// TIA Portal V17 export
// export: Created 2026-04-13T11:12:41.7444866Z, ExportSetting WithDefaults, DisplayName Totally Integrated Automation Portal, DisplayVersion V17 Update 4, DisplayName TIA Portal Openness, DisplayVersion V17 Update 4, DisplayName TIA Portal Version Control Interface, DisplayVersion V17, DisplayName SINAMICS Startdrive Advanced, DisplayVersion V17, DisplayName SINAMICS Startdrive G130, G150, S120, S150, SINAMICS MV, S210, DisplayVersion V17, DisplayName SINAMICS Startdrive G110M, G120, G120C, G120D, G120P, G115D, DisplayVersion V17, DisplayName STEP 7 Professional, DisplayVersion V17 Update 4, DisplayName STEP 7 Safety, DisplayVersion V17, DisplayName WinCC Professional, DisplayVersion V17 Update 4
FUNCTION_BLOCK "A9-循环下料控制"   // FB15, SCL
{ S7_Optimized_Access := 'TRUE' }
VERSION : 0.1
// stored: AutoNumber true, IsIECCheckEnabled false, IsRetainMemResEnabled false, MemoryReserve 100, SetENOAutomatically false, UDAEnableTagReadback false
   VAR_INPUT
      下料启动开关 : Bool;
      上卸料阀工作时间 : Real;
      上卸料阀关闭时间 : Real;
      下卸料阀工作时间 : Real;
      下卸料阀关闭时间 : Real;
   END_VAR
   VAR_OUTPUT
      上阀实际工作时间 : Real;
      上阀实际停止时间 : Real;
      下阀实际工作时间 : Real;
      下阀实际停止时间 : Real;
   END_VAR
   VAR_IN_OUT
      上下料阀 : Bool;
      下下料阀 : Bool;
      振动筛 : Bool;
   END_VAR
   VAR
      上下料阀实际工作时间 : Time;
      上下料阀实际停止时间 : Time;
      下下料阀实际工作时间 : Time;
      下下料阀实际停止时间 : Time;
      循环间隔实际时间 : Time;
      上阀打开辅助 : Bool;
      上阀关闭辅助 : Bool;
      下阀打开辅助 : Bool;
      下阀关闭辅助 : Bool;
      循环工作时间延时 { S7_SetPoint := 'True'} : TON_TIME;
      上阀打开检测1 { S7_SetPoint := 'True'} : R_TRIG;
      上阀打开检测2 { S7_SetPoint := 'True'} : R_TRIG;
      上阀工作时间延时 { S7_SetPoint := 'True'} : TON_TIME;
      上阀停止时间延时 { S7_SetPoint := 'True'} : TON_TIME;
      下阀工作时间延时 { S7_SetPoint := 'True'} : TON_TIME;
      下阀停止时间延时 { S7_SetPoint := 'True'} : TON_TIME;
      下阀打开检测 { S7_SetPoint := 'True'} : R_TRIG;
   END_VAR
BEGIN

   #上下料阀实际工作时间 := DINT_TO_TIME(REAL_TO_DINT(#上卸料阀工作时间*1000.0));
   #上下料阀实际停止时间 := DINT_TO_TIME(REAL_TO_DINT(#上卸料阀关闭时间 * 1000.0));
   #下下料阀实际工作时间 := DINT_TO_TIME(REAL_TO_DINT(#下卸料阀工作时间 * 1000.0));
   #下下料阀实际停止时间 := DINT_TO_TIME(REAL_TO_DINT(#下卸料阀关闭时间 * 1000.0));

   #上阀打开检测1(CLK:=#下料启动开关);


   IF #上阀打开检测1.Q THEN
       #上阀打开辅助 := TRUE;
   END_IF;


   #上阀工作时间延时.TON(IN:=#上阀打开辅助 AND #下料启动开关 AND NOT #下阀停止时间延时.Q,PT:=#上下料阀实际工作时间);

   #上阀停止时间延时.TON(IN:=#上阀工作时间延时.Q,PT:=#上下料阀实际停止时间);

   #下阀工作时间延时(IN:=#上阀工作时间延时.Q AND #上阀停止时间延时.Q,PT:=#下下料阀实际工作时间);

   #下阀停止时间延时(IN :=#上阀工作时间延时.Q AND #上阀停止时间延时.Q AND  #下阀工作时间延时.Q,PT := #下下料阀实际停止时间);

   #下阀打开检测(CLK:=#下下料阀);


   #上下料阀 := #上阀打开辅助 AND NOT #上阀工作时间延时.Q AND #下料启动开关;


   #下下料阀 := #上阀工作时间延时.Q AND #上阀停止时间延时.Q AND NOT #下阀工作时间延时.Q AND #下料启动开关;

   IF #下阀打开检测.Q AND #下料启动开关 THEN
       #振动筛 := true;
   END_IF;

   IF NOT #下料启动开关 THEN
       #上阀打开辅助 := false;
   END_IF;

   IF #上下料阀 THEN
       #上阀实际工作时间 := DINT_TO_REAL(TIME_TO_DINT(#上阀工作时间延时.ET))/1000.0;
   END_IF;

   IF #上阀工作时间延时.Q AND NOT #上阀停止时间延时.Q THEN
       #上阀实际停止时间 := DINT_TO_REAL(TIME_TO_DINT(#上阀停止时间延时.ET)) / 1000.0;
   END_IF;

   IF #下下料阀 THEN
       #下阀实际工作时间 := DINT_TO_REAL(TIME_TO_DINT(#下阀工作时间延时.ET)) / 1000.0;
   END_IF;

   IF #下阀工作时间延时.Q AND NOT #下阀停止时间延时.Q THEN
       #下阀实际停止时间 := DINT_TO_REAL(TIME_TO_DINT(#下阀停止时间延时.ET)) / 1000.0;
   END_IF;
END_FUNCTION_BLOCK
